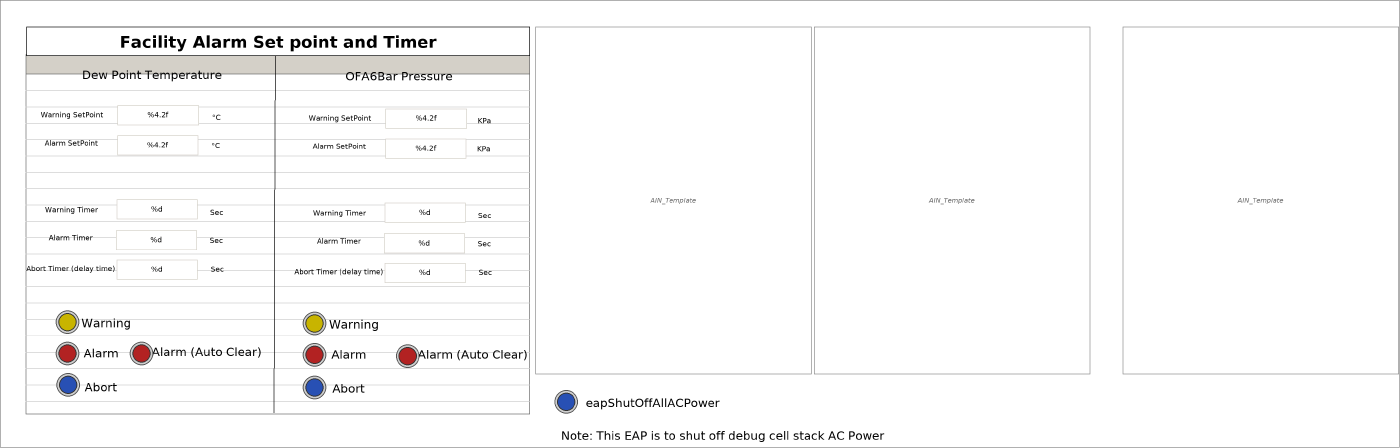
VISUALIZATION HMI_FacilityAlarm_OFADewpoint  // 2136x685
    Table (39,83 769x550)
    Rectangle (40,41 768x44)
    Label (48,49 753x30), "Facility Alarm Set point and Timer"
    Label (41,90 382x50), "Dew Point Temperature"
    Label (421,92 376x50), "OFA6Bar Pressure"
    Line (418,631) (420,85)
    Textfield (179,161 124x30), "%4.2f", text variable: DewPoint_LowSP
        OnMouseClick: write DewPoint_LowSP via Default
    Label (44,161 132x30), "Warning SetPoint"
    Label (308,165 44x30), "°C"
    Label (43,204 132x30), "Alarm SetPoint"
    Textfield (179,207 123x30), "%4.2f", text variable: DewPoint_LowLowSP
        OnMouseClick: write DewPoint_LowLowSP via Default
    Label (307,208 44x30), "°C"
    Textfield (178,305 123x30), "%d", text variable: DewPoint_Warning_Timer
        OnMouseClick: write DewPoint_Warning_Timer via Default
    Label (42,306 134x30), "Warning Timer"
    Label (306,310 49x30), "Sec"
    Textfield (177,352 123x30), "%d", text variable: DewPoint_Alarm_Timer
        OnMouseClick: write DewPoint_Alarm_Timer via Default
    Label (41,349 134x30), "Alarm Timer"
    Label (305,353 50x30), "Sec"
    Textfield (178,397 123x30), "%d", text variable: DewPoint_Abort_Timer
        OnMouseClick: write DewPoint_Abort_Timer via Default
    Label (42,396 132x30), "Abort Timer (delay time)"
    Label (305,397 53x30), "Sec"
    Label (453,166 132x30), "Warning SetPoint"
    Textfield (588,166 124x30), "%4.2f", text variable: OFA6Bar_LowSP
        OnMouseClick: write OFA6Bar_LowSP via Default
    Label (717,170 44x30), "KPa"
    Label (452,209 132x30), "Alarm SetPoint"
    Textfield (588,212 123x30), "%4.2f", text variable: OFA6Bar_LowLowSP
        OnMouseClick: write OFA6Bar_LowLowSP via Default
    Label (716,213 44x30), "KPa"
    Textfield (587,310 123x30), "%d", text variable: OFA6Bar_Warning_Timer
        OnMouseClick: write OFA6Bar_Warning_Timer via Default
    Label (451,311 134x30), "Warning Timer"
    Label (715,315 49x30), "Sec"
    Textfield (586,357 123x30), "%d", text variable: OFA6Bar_Alarm_Timer
        OnMouseClick: write OFA6Bar_Alarm_Timer via Default
    Label (450,354 134x30), "Alarm Timer"
    Label (714,358 50x30), "Sec"
    Textfield (587,402 123x30), "%d", text variable: OFA6Bar_Abort_Timer
        OnMouseClick: write OFA6Bar_Abort_Timer via Default
    Label (451,401 132x30), "Abort Timer (delay time)"
    Label (714,402 53x30), "Sec"
    Frame (817,41 421x531)
        shows AIN_Template(DUT := fbDebugColumn.fb_facility_DewPoint_OFA6Bar._DUT_AIN_InletTemp)
    Frame (1242,41 421x531)
        shows AIN_Template(DUT := fbDebugColumn.fb_facility_DewPoint_OFA6Bar._DUT_AIN_DewPoint)
    Frame (1713,41 421x531)
        shows AIN_Template(DUT := fbDebugColumn.fb_facility_DewPoint_OFA6Bar._DUT_AIN_6BarOFA)
    Lamp1 (77,472 52x41), variable: ALM_DCCOL.AlarmID[15], style: Lamp-Lamp1-Yellow
    Lamp1 (77,520 52x41), variable: ALM_DCCOL.AlarmID[4], style: Lamp-Lamp1-Red
    Lamp1 (454,522 52x41), variable: ALM_DCCOL.AlarmID[5], style: Lamp-Lamp1-Red
    Lamp1 (454,474 52x41), variable: ALM_DCCOL.AlarmID[12], style: Lamp-Lamp1-Yellow
    Label (491,480 98x33), "Warning"
    Label (493,526 79x33), "Alarm"
    Lamp1 (454,572 52x41), variable: OFA6Bar_Abort, style: Lamp-Lamp1-Blue
    Label (491,578 82x33), "Abort"
    Lamp1 (78,568 52x41), variable: DewPoint_Abort, style: Lamp-Lamp1-Blue
    Lamp1 (838,594 52x41), variable: fbDebugColumn.stDebugColumnDIO.eapShutOffAllACPower, style: Lamp-Lamp1-Blue
    Label (875,600 242x33), "eapShutOffAllACPower"
    Label (824,650 557x33), "Note: This EAP is to shut off debug cell stack AC Power"
    Label (113,478 98x33), "Warning"
    Label (115,524 79x33), "Alarm"
    Label (113,576 82x33), "Abort"
    Label (635,526 173x33), "Alarm (Auto Clear)"
    Lamp1 (596,524 52x41), variable: OFA6Bar_Alarm, style: Lamp-Lamp1-Red
    Label (229,522 173x33), "Alarm (Auto Clear)"
    Lamp1 (190,520 52x41), variable: DewPoint_Alarm, style: Lamp-Lamp1-Red
END_VISUALIZATION

(* stored: Version 1.1.0.1, ProductVersion 3.1.4022.18
   Visu HMI_FacilityAlarm_OFADewpoint: Id {a36eeb12-0ad8-487f-a2c1-f14ce10616f4} *)
